Staubli VAL3: action_buffer.pgx

program action_buffer()
  local ActionItem l_aAction
  local bool l_bEmpty
begin
  // wait the Task Cycle or simulation has been started
  wait(cycleStatus:bCycle or cycleStatus:bSimulation)
  //
  // scan the action
  //
  while (cycleStatus:bCycle or cycleStatus:bSimulation)
    // wait to move to run STATE
    do
      // scan the action item
      call cycleStatus:isActionEmpty(l_bEmpty)
      cycleStatus:bActionRunning=!l_bEmpty
      if !(cycleStatus:bCycle or cycleStatus:bSimulation)
        return
      endIf
      delay(0)
    until l_bEmpty==false
    // execute
    call cycleStatus:getAction(l_aAction)
    call action_do(l_aAction,-1)
    // remove
    call cycleStatus:removeAction()
  endWhile
  //
end
